// TIA Portal V20 export
FUNCTION "StepToString" : String   // FC88, SCL
// stored: Namespace Unit1.Em5, SetENOAutomatically false
   VAR_INPUT
      StepDINT : DInt;   // DINT value of the step
   END_VAR
BEGIN
   // Translates the sequence step number to the step name
   // Adjusted for Sequence_1_ManualInput real use case

   CASE #StepDINT OF
       1:
           #StepToString := 'Idle';

       101:
           #StepToString := 'JOB[1] Condition';
       111:
           #StepToString := 'Cylinder HomePos & Magazine Lock WorkPos Check';
       121:
           #StepToString := 'Vacuum HomePos & Vibrator HomePos Check';
       131:
           #StepToString := 'AxisY & Magazine AxisZ Homed Check';
       141:
           #StepToString := 'AxisY & Magazine AxisZ HomePos Check';
       151:
           #StepToString := 'Magazine AxisZ PickUpPos Check';
       191:
           #StepToString := 'JOB[1] Step End';

       201:
           #StepToString := 'JOB[2] Condition';
       211:
           #StepToString := 'Cylinder WorkPos Command';
       221:
           #StepToString := 'Vacuum WorkPos Command';
       231:
           #StepToString := 'Vibrator WorkPos Command';
       241:
           #StepToString := 'Magazine AxisZ EvasionPos Command';
       251:
           #StepToString := 'Vibrator HomePos Command';
       261:
           #StepToString := 'Cylinder HomePos Command';
       291:
           #StepToString := 'JOB[2] Step End';

       301:
           #StepToString := 'JOB[3] Condition';
       311:
           #StepToString := 'AxisY ConveyorPos Command';
       321:
           #StepToString := 'Cylinder WorkPos Command';
       331:
           #StepToString := 'Vacuum HomePos Command';
       341:
           #StepToString := 'Cylinder HomePos Command';
       351:
           #StepToString := 'AxisY HomePos Command';
       391:
           #StepToString := 'JOB[3] Step End';

       901:
           #StepToString := 'Immediate Stop';

       ELSE
           #StepToString := 'N/A';

   END_CASE;
END_FUNCTION
